{attribute addProperty BoxType "AT2050-0500-0021"}
{attribute addProperty Id "A_0092_AT2020_5250_0018_AT2020_5250AT2020_C5E5984862678.25"}
{attribute addProperty CRC "692802805"}
{attribute addProperty SizeInBites "626"}
{attribute addProperty SizeInBytes "78.25"}
TYPE A_0052_AT2050_0500_0021_294B54F5 EXTENDS AT2050_BA5A9548 :
STRUCT
	{attribute addProperty Name "A_0092_AT2020_5250_0018_AT2020_5250"}
	A_0092_AT2020_5250_0018_AT2020_5250 : AT2020_C5E59848;
END_STRUCT
END_TYPE

(* stored: Version 1.2.0.0, ProductVersion 3.1.4024.9
   DUT A_0052_AT2050_0500_0021_294B54F5: Id {90a8bf47-512b-4f7b-a1f6-bc2c2fdefefb} *)
